Staubli VAL3: default.pjx

Parameters version=s8.5.4cs9_BS1251 stackSize=5000 millimeterUnit=true
Program file=start.pgx
Program file=stop.pgx
Data file=default.dtx
